/// configuration data that is used during boot to configure the Units equipment
TYPE ScriblyDataConfig :
STRUCT
  Simulated : BOOL;
END_STRUCT
END_TYPE

(* stored: Version 1.1.0.1
   DUT ScriblyDataConfig: Id {58c8b0c9-4d05-4c04-abf4-f23facd36340} *)
